FUNCTION_BLOCK RequestOrchestrationHTTP (* Request Orchestration Function Block using HTTP *)
  (* Standard: 61499-2; Description: Copyright (c) 2018 fortiss GmbH This program and the accompanying materials are made available under the terms of the Eclipse Public License 2.0 which is available at https://www.eclipse.org/legal/epl-2.0/ SPDX-License-Identifier: EPL-2.0 *)
  (* Version 1.0, 2018-09-21, Jose Cabral, fortiss GmbH *)
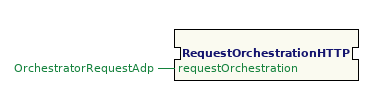
  SOCKETS
    requestOrchestration : OrchestratorRequestAdp; (* Request orchestration adapter *)
  END_SOCKETS
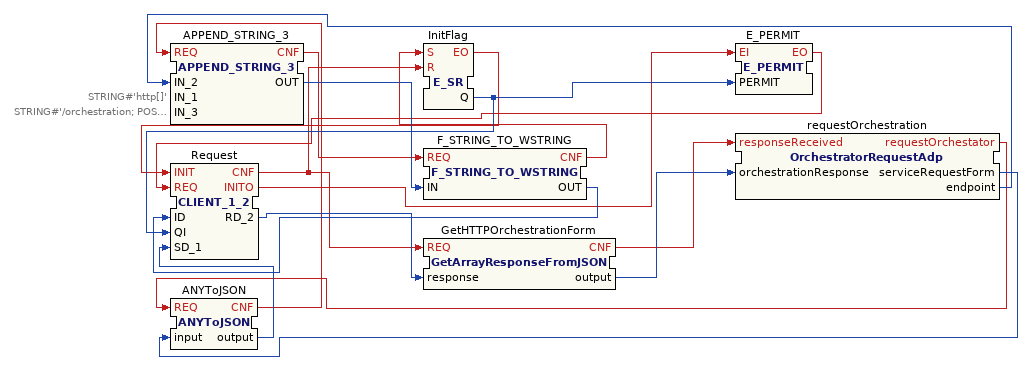
  FBS
    APPEND_STRING_3 : APPEND_STRING_3(IN_1 := STRING#'http[]', IN_3 := STRING#'/orchestration; POST; application/json]');
    Request : CLIENT_1_2;
    InitFlag : E_SR;
    E_PERMIT : E_PERMIT;
    F_STRING_TO_WSTRING : F_STRING_TO_WSTRING;
    ANYToJSON : ANYToJSON;
    GetHTTPOrchestrationForm : GetArrayResponseFromJSON;
  END_FBS
  EVENT_CONNECTIONS
    APPEND_STRING_3.CNF TO F_STRING_TO_WSTRING.REQ;
    F_STRING_TO_WSTRING.CNF TO InitFlag.S;
    InitFlag.EO TO Request.INIT;
    E_PERMIT.EO TO Request.REQ;
    ANYToJSON.CNF TO APPEND_STRING_3.REQ;
    Request.CNF TO InitFlag.R;
    Request.INITO TO E_PERMIT.EI;
    requestOrchestration.requestOrchestator TO ANYToJSON.REQ;
    Request.CNF TO GetHTTPOrchestrationForm.REQ;
    GetHTTPOrchestrationForm.CNF TO requestOrchestration.responseReceived;
  END_CONNECTIONS
  DATA_CONNECTIONS
    APPEND_STRING_3.OUT TO F_STRING_TO_WSTRING.IN;
    F_STRING_TO_WSTRING.OUT TO Request.ID;
    InitFlag.Q TO E_PERMIT.PERMIT;
    InitFlag.Q TO Request.QI;
    ANYToJSON.output TO Request.SD_1;
    requestOrchestration.serviceRequestForm TO ANYToJSON.input;
    requestOrchestration.endpoint TO APPEND_STRING_3.IN_2;
    Request.RD_2 TO GetHTTPOrchestrationForm.response;
    GetHTTPOrchestrationForm.output TO requestOrchestration.orchestrationResponse;
  END_CONNECTIONS
END_FUNCTION_BLOCK
